SUBAPPLICATION Vorsteuerventil (* Subapplication Type *)
  (* Standard: 61499-2 *)
  (* Version 1.0, 2023-01-29, Franz *)
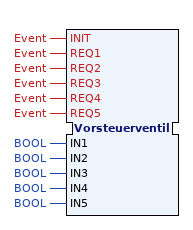
  EVENT_INPUT
    INIT;
    REQ1;
    REQ2;
    REQ3;
    REQ4;
    REQ5;
  END_EVENT
  VAR_INPUT
    IN1 : BOOL;
    IN2 : BOOL;
    IN3 : BOOL;
    IN4 : BOOL;
    IN5 : BOOL;
  END_VAR
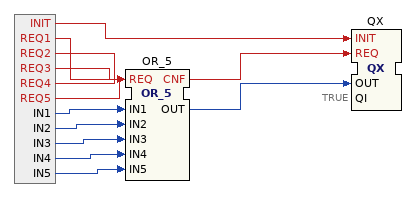
  FBS
    OR_5 : OR_5;
    QX : QX(QI := TRUE);
  END_FBS
  EVENT_CONNECTIONS
    REQ1 TO OR_5.REQ;
    REQ2 TO OR_5.REQ;
    REQ3 TO OR_5.REQ;
    REQ4 TO OR_5.REQ;
    REQ5 TO OR_5.REQ;
    INIT TO QX.INIT;
    OR_5.CNF TO QX.REQ;
  END_CONNECTIONS
  DATA_CONNECTIONS
    IN1 TO OR_5.IN1;
    IN2 TO OR_5.IN2;
    IN3 TO OR_5.IN3;
    IN4 TO OR_5.IN4;
    IN5 TO OR_5.IN5;
    OR_5.OUT TO QX.OUT;
  END_CONNECTIONS
END_SUBAPPLICATION
